// TIA Portal V16 export
// export: Created 2021-11-12T13:33:10.6819299Z, ExportSetting WithDefaults, DisplayName Totally Integrated Automation Portal, DisplayVersion V16 Update 3, DisplayName TIA Portal Version Control Interface, DisplayVersion V16 Update 2, DisplayName TIA Portal Openness, DisplayVersion V16 Update 3, DisplayName SINAMICS Startdrive Advanced, DisplayVersion V16 Update 5, DisplayName SINAMICS Startdrive G130, G150, S120, S150, SINAMICS MV, S210, DisplayVersion V16 Update 5, DisplayName SINAMICS Startdrive G110M, G120, G120C, G120D, G120P, G115D, DisplayVersion V16 Update 5, DisplayName STEP 7 Professional, DisplayVersion V16 Update 3, DisplayName STEP 7 Safety, DisplayVersion V16, DisplayName WinCC UA Professional, DisplayVersion V16 Update 3
DATA_BLOCK "HMI_CMD_450"   // DB96
{ S7_Optimized_Access := 'TRUE' }
VERSION : 0.1
// stored: AutoNumber true, DBAccessibleFromOPCUA true, IsOnlyStoredInLoadMemory false, IsRetainMemResEnabled false, IsWriteProtectedInAS false, MemoryReserve 100
   VAR
      xxxxx___BinarySensors___xxxxx : Byte;
      "GL01-BG01" : "UDT_CH_DI_Command";   // Reflexní optická závora - Snímání pohybu dílu na dopravníku
      "GL02-BG01" : "UDT_CH_DI_Command";   // Reflexní optická závora - Snímání pohybu dílu na dopravníku
      "GL03-BG01" : "UDT_CH_DI_Command";   // Reflexní optická závora - Snímání pohybu dílu na dopravníku
      "GL04-BG01" : "UDT_CH_DI_Command";   // Reflexní optická závora - Snímání pohybu dílu na dopravníku
      "UC21-FC01_14" : "UDT_CH_DI_Command";   // 400V Dopravník ++450 OK
      "UC21-FC02_14" : "UDT_CH_DI_Command";   // 400V Dopravník ++450 OK
      "UC21-FC03_14" : "UDT_CH_DI_Command";   // 400V Dopravník ++450 OK
      "UC21-FC04_14" : "UDT_CH_DI_Command";   // 400V Dopravník ++450 OK
      "GL01-BG01_4" { S7_SetPoint := 'True'} : "UDT_CH_DI_Command";   // Snímání pohybu dílu na dopravníku ++450+GL01 (M2)
      "GL02-BG01_4" { S7_SetPoint := 'True'} : "UDT_CH_DI_Command";   // Snímání pohybu dílu na dopravníku ++450+GL02 (M4)
      "GL03-BG01_4" { S7_SetPoint := 'True'} : "UDT_CH_DI_Command";   // Snímání pohybu dílu na dopravníku ++450+GL03 (M7.1)
      "GL04-BG01_4" { S7_SetPoint := 'True'} : "UDT_CH_DI_Command";   // Snímání pohybu dílu na dopravníku ++450+GL04 (M6)
      xxxxx___BinaryOthers___xxxxx : Byte;
      "UH11-SF01_14" : "UDT_CH_DI_Command";   // Conveyor Remote
      "UH11-SF01_24" : "UDT_CH_DI_Command";   // Conveyor Automat
      "UH11-SF03_14" : "UDT_CH_DI_Command";   // Conveyor Start automat
      "UH11-SF04_12" : "UDT_CH_DI_Command";   // Conveyor Stop
      "UH11-SF05_14" : "UDT_CH_DI_Command";   // Conveyor GL02 Manual Backward
      "UH11-SF05_24" : "UDT_CH_DI_Command";   // Conveyor GL02 Manual Forward
      "UH11-SF06_14" : "UDT_CH_DI_Command";   // Conveyor GL03 Manual Backward
      "UH11-SF06_24" : "UDT_CH_DI_Command";   // Conveyor GL03 Manual Forward
      "UH11-SF07_14" : "UDT_CH_DI_Command";   // Conveyor GL04 Manual Backward
      "UH11-SF07_24" : "UDT_CH_DI_Command";   // Conveyor GL04 Manual Forward
      "UH11-SF08_14" : "UDT_CH_DI_Command";   // Bedna Žádost o výměnu
      "UH11-SF09_14" : "UDT_CH_DI_Command";   // Bedna vyměněna
      "UH31-SF02_14" { S7_SetPoint := 'True'} : "UDT_CH_DI_Command";   // Conveyor GL01 Remote
      "UH31-SF02_24" { S7_SetPoint := 'True'} : "UDT_CH_DI_Command";   // Conveyor GL01 Automat
      "UH31-SF04_14" { S7_SetPoint := 'True'} : "UDT_CH_DI_Command";   // Conveyor GL01 Start automat
      "UH31-SF03_14" { S7_SetPoint := 'True'} : "UDT_CH_DI_Command";   // Conveyor GL01 Manual Backward
      "UH31-SF03_24" { S7_SetPoint := 'True'} : "UDT_CH_DI_Command";   // Conveyor GL01 Manual Forward
      "UH31-SF06_X2" { S7_SetPoint := 'True'} : "UDT_CH_DI_Command";   // Dopravník GL01 - blokování pásu v peci
      "UH31-SF05_12" { S7_SetPoint := 'True'} : "UDT_CH_DI_Command";   // Conveyor GL01 Stop
      GL03_PartsToBox { S7_SetPoint := 'True'} : Bool;   // Send all parts to box
      xxxxx___Drives___xxxxx : Byte;
      "GL01-MA01" : "UDT_Drive1_Command";   // Dopravník ke tryskači (M2)
      "GL02-MA01" : "UDT_Drive1_Command";   // Dopravník ke tryskači (M4)
      "GL03-MA01" : "UDT_Drive1_Command";   // Dopravník ke tryskači (M7.1)
      "GL04-MA01" : "UDT_Drive1_Command";   // Dopravník ke tryskači (M6)
      "UC21-TA01" : "UDT_SINAMICS_G120_Command";   // Měnič
      "UC21-TA02" : "UDT_SINAMICS_G120_Command";   // Měnič
      "UC21-TA03" : "UDT_SINAMICS_G120_Command";   // Měnič
      "UC21-TA04" : "UDT_SINAMICS_G120_Command";   // Měnič
      xxxxx___Others___xxxxx : Byte;
      CL01 : "UDT_PartCounter_Command";   // Box
      xxxxx___Alarms___xxxxx : Byte;
      CL01_Alarm : "UDT_DI_Mon_Command";   // CL01 - box full alarm
      CL01_Warn : "UDT_DI_Mon_Command";   // CL01 - box full warning
   END_VAR
BEGIN
END_DATA_BLOCK
